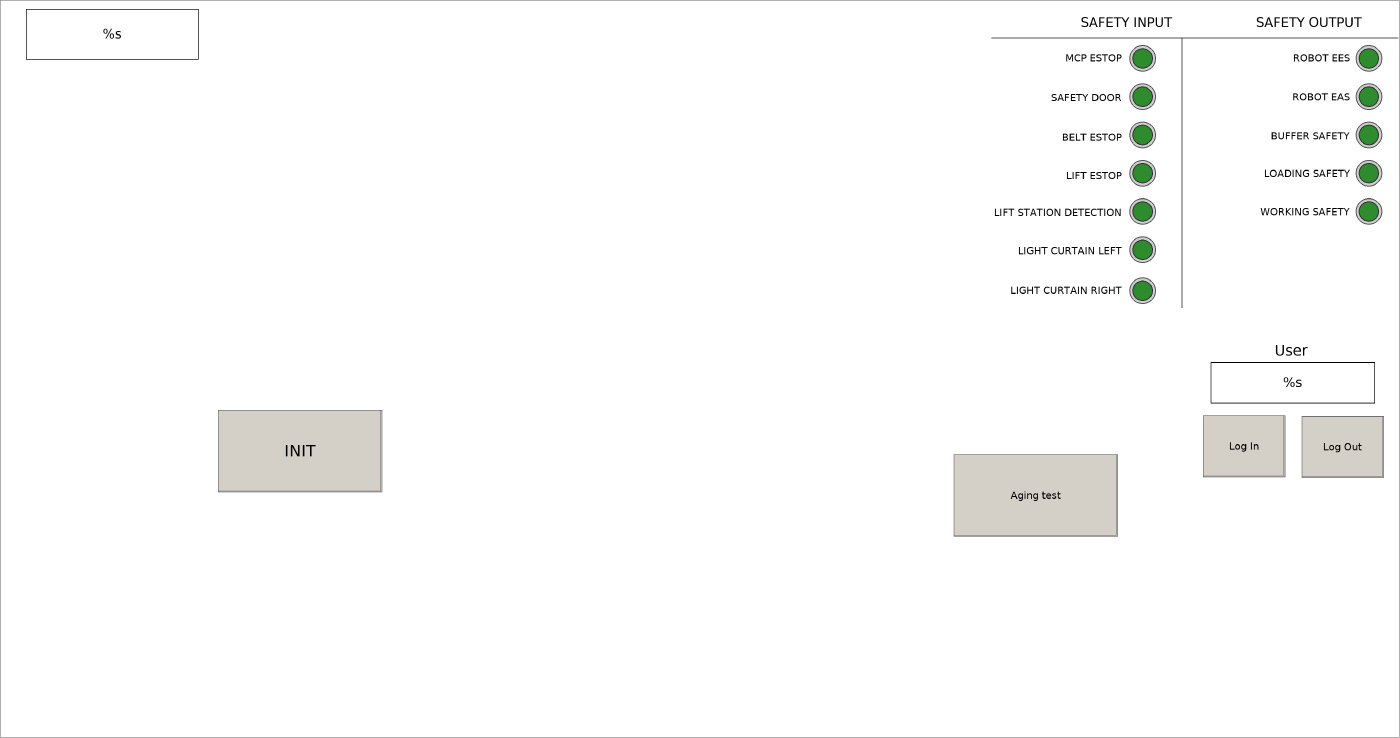
VISUALIZATION visu_operation  // 2048x1080
    Button (319,600 240x120), "INIT", colour toggle: G_HMI.bInit
        OnMouseDown: execute { G_HMI.bInit	:= TRUE; }
        OnMouseUp: execute { G_HMI.bInit	:= FALSE; }
    Lamp1 (1649,63 45x45), variable: MAIN.application.safety.mcp_estop, style: Lamp-Lamp1-Green
    Label (1344,70 300x30), "MCP ESTOP"
    Lamp1 (1649,175 45x45), variable: MAIN.application.safety.belt_estop, style: Lamp-Lamp1-Green
    Label (1344,186 300x30), "BELT ESTOP"
    Lamp1 (1649,231 45x45), variable: MAIN.application.safety.lift_estop, style: Lamp-Lamp1-Green
    Label (1344,244 300x26), "LIFT ESTOP"
    Lamp1 (1649,287 45x45), variable: MAIN.application.safety.lift_station_detection, style: Lamp-Lamp1-Green
    Label (1344,298 300x26), "LIFT STATION DETECTION"
    Lamp1 (1649,119 45x45), variable: MAIN.application.safety.mcp_safetyDoor, style: Lamp-Lamp1-Green
    Label (1344,128 300x30), "SAFETY DOOR"
    Lamp1 (1649,343 45x45), variable: MAIN.application.safety.lift_lightCurtain_left, style: Lamp-Lamp1-Green
    Label (1344,352 300x30), "LIGHT CURTAIN LEFT"
    Lamp1 (1649,403 45x45), variable: MAIN.application.safety.lift_lightCurtain_right, style: Lamp-Lamp1-Green
    Label (1344,410 300x30), "LIGHT CURTAIN RIGHT"
    Lamp1 (1980,63 45x45), variable: MAIN.application.safety.robot_EES, style: Lamp-Lamp1-Green
    Label (1728,70 250x30), "ROBOT EES"
    Lamp1 (1980,175 45x45), variable: MAIN.application.safety.buffer_safety, style: Lamp-Lamp1-Green
    Label (1728,184 250x30), "BUFFER SAFETY"
    Lamp1 (1980,231 45x45), variable: MAIN.application.safety.loading_safety, style: Lamp-Lamp1-Green
    Label (1728,241 250x26), "LOADING SAFETY"
    Lamp1 (1980,287 45x45), variable: MAIN.application.safety.working_safety, style: Lamp-Lamp1-Green
    Label (1728,297 250x26), "WORKING SAFETY"
    Lamp1 (1980,119 45x45), variable: MAIN.application.safety.robot_EAS, style: Lamp-Lamp1-Green
    Label (1728,127 250x30), "ROBOT EAS"
    Line (1729,450) (1729,55)
    Label (1523,18 250x30), "SAFETY INPUT"
    Label (1790,18 250x30), "SAFETY OUTPUT"
    Line (1450,55) (2045,55)
    Button (1395,665 240x120), "Aging test", colour toggle: G_HMI.bAging_test
        toggle G_HMI.bAging_test
    Rectangle (38,13 252x74), "%s"
    Rectangle (1771,530 240x60), "%s", text variable: G_HMI.sLoginnedUser
    Button (1904,609 120x90), "Log Out"
        OnMouseDown: VisuUserMgmt Type=Logout
    Button (1760,608 120x90), "Log In"
        OnMouseDown: VisuUserMgmt Type=Login
    Label (1814,498 150x30), "User"
END_VISUALIZATION

(* stored: Version 1.1.0.1, ProductVersion 3.1.4024.12
   Visu visu_operation: Id {4abbf3f6-c173-4bcb-82b6-c0f3163ef68d} *)
